(* PLC project ap_master, Dassault Systèmes ControlBuild 2024x Refresh1 *)
(* stored: creationDateTime 2024-04-12T15:10:27-01:00 *)

PROGRAM ap_master.ap_master

(* FBD diagram, written out as Structured Text *)
END_PROGRAM
